TYPE ST_InputConvData :
STRUCT
	id :INT;
	timeStampin :STRING;
	timeStamparrived:STRING;
	timeStampout:STRING;
END_STRUCT
END_TYPE

(* stored: Version 1.1.0.1, ProductVersion 3.1.4026.17
   DUT ST_InputConvData: Id {379253df-0555-410e-8cde-272d7d813f36} *)
